(* PLC project 06_ld_pool.project, CODESYS CODESYS V3.5 SP22 Patch 3 *)
(* stored: creationDateTime 2026-09-21T20:53:57.7515587, modificationDateTime 2026-09-21T20:35:18.3594477 *)

VAR_GLOBAL  (* GVL_Pool *)
  gPoolCount : INT;
  gPoolFlag : BOOL;
END_VAR

FUNCTION_BLOCK FB_PoolUser
  VAR_EXTERNAL
    gPoolCount : INT;
  END_VAR
  VAR_OUTPUT
    xFlagSeen : BOOL;
  END_VAR

            gPoolCount := gPoolCount + 1;
xFlagSeen := GVL_Pool.gPoolFlag;
          
END_FUNCTION_BLOCK

PROGRAM PLC_PRG
  VAR
    fbPool : FB_PoolUser;
    bHorn : BOOL;
    bDoorClosed : BOOL;
    bLampRun : BOOL;
  END_VAR

                    PRG_Ladder();
fbPool();
IF (bHorn S= bDoorClosed) THEN bLampRun := TRUE; END_IF;
                  
END_PROGRAM

PROGRAM PRG_Ladder
  VAR
    xStart : BOOL;
    xDone : BOOL;
    xLamp : BOOL;
    iCount : INT;
    tonDelay : TON;
    tElapsed : TIME;
  END_VAR

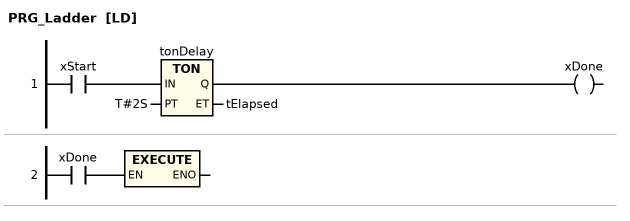
(* LD diagram, written out as Structured Text *)

tonDelay(IN := xStart, PT := T#2S, ET => tElapsed);
xDone := tonDelay.Q;

IF xDone THEN
  iCount := iCount + 1;
     xLamp := xDone AND xStart;
END_IF;
END_PROGRAM

CONFIGURATION Device
  RESOURCE Application ON PLC
    TASK MainTask(INTERVAL := T#20ms, PRIORITY := 1);
    PROGRAM PLC_PRG WITH MainTask : PLC_PRG;
  END_RESOURCE
END_CONFIGURATION
